(* PLC project v0.6.04_CycleSemiAuto.project, CODESYS CODESYS V3.5 SP19 Patch 1 *)
(* stored: creationDateTime 2026-08-04T14:33:45.723569, modificationDateTime 2026-08-04T14:33:45.723569 *)

(* ═══════════════════════════════════════════════════════════════ 🧲 ST_EncoderHMI — Données d'échange IHM pour les codeurs absolus ─────────────────────────────────────────────────────────────── 🎨 Destiné à l'affichage des informations et diagnostics des codeurs. ═══════════════════════════════════════════════════════════════ *)
TYPE ST_EncoderHMI : STRUCT
  RawPos : UDINT;  (* 📊 Position brute lue sur le bus *)
  Alarms : UINT;  (* ⚠️ Code d'alarme brut du codeur *)
  Warnings : UINT;  (* 🟧 Code d'avertissement brut du codeur *)
  SlaveOperational : BOOL;  (* 📡 Esclave EtherCAT opérationnel *)
  PresetTriggerCmd : WORD;  (* 🎯 Commande de preset active *)
  PresetValueOut : UDINT;  (* 📐 Valeur de preset envoyée au codeur *)
  Error : BOOL;  (* 🔴 Codeur en défaut (liaison EtherCAT ou preset) *)
  ErrorId : WORD;  (* ❌ Code défaut codeur *)
  Homed : BOOL;  (* 🎯 Homing — déplacés depuis ST_WinchState racine (2026-08, réorganisation ST_WinchHMI/Homing) 🎯 Prise d'origine (Homing) validée *)
  HomingBusy : BOOL;  (* ⏳ Référencement en cours *)
  HomingDone : BOOL;  (* ✅ Pulse de référencement réussi *)
  HomingError : BOOL;  (* 🔴 Défaut de référencement *)
  HomingErrorId : WORD;  (* ❌ Bitfield défaut homing *)
  HomingState : E_State;  (* 🤖 État FB_Encoder_Homing *)
  HomingStateAtError : E_State;  (* 🧭 État lors du défaut *)
  HomingSuspect : BOOL;  (* ⚠️ Référence à confirmer *)
  HomingRefRaw : UDINT;  (* 📐 Référence brute appliquée *)
END_STRUCT;
END_TYPE

(* values of E_State: DISABLED: Enable faux, neutralisé; INIT: Démarrage / vérifs; READY: Prêt, attend ordre; BUSY: Action en cours; DONE: Action terminée; STOPPING: Décél rampe avant arrêt (StartStop=FALSE ou SafeStop=TRUE) *)

{attribute 'qualified_only'}
{attribute 'strict'}
TYPE E_State : (DISABLED := 0, INIT := 1, READY := 2, BUSY := 3, DONE := 4, STOPPING := 5);
END_TYPE
